{attribute 'Tc2GvlVarNames'}
VAR_GLOBAL
END_VAR

(* stored: Version 1.1.0.1, ProductVersion 3.1.4024.9
   GVL Globale_Variablen: Id {86ef11db-5491-4217-bde7-ad4fe417abb1} *)
